(*
SPDX-FileCopyrightText: © 2026 Oleksandr Tiutyk <trofimich@gmail.com>
SPDX-License-Identifier: MIT
License: https://opensource.org/license/mit
*)

INTERFACE IIncompartibleGenericValueTypeException EXTENDS IGeneralException

METHOD Throw
VAR_INPUT
	sourceNamespaceName : STRING;
	sourceClassName : STRING;
	sourcePOUName : STRING;
	sourcePosition : STRING;
	validatedObjectName : WSTRING;
	actualTypeClass : GENERIC_TYPE_CLASS;
	expectedTypeClass : GENERIC_TYPE_CLASS;
END_VAR
END_METHOD

END_INTERFACE

(* stored: Version 1.1.0.1
   Itf IIncompartibleGenericValueTypeException: Id {feeaa4aa-5b5e-462e-9c3e-1501eb3608c2}
   Method Throw: Id {bfb374d5-a64b-4d06-8c34-af2cdfea1228} *)
